TYPE DUT_HMI_06 :
STRUCT
	Manuals : DUT_HMI_06_MANUALS;
	ProductStatus 	: eProductStatus;
	State			: eStationState;
	EVDiagnostic 	: ARRAY[0..20] OF DUT_HMI_EV_Diagnostic;
	EVInfo			: ARRAY[0..CNC.NUM_MAX_MANUALS_06-1] OF DUT_HMI_EV_Info;
	Status			: USINT;
	CycleTime		: STRING;
	BroachTarget	: USINT;
END_STRUCT
END_TYPE

(* stored: Version 1.1.0.1, ProductVersion 3.1.4024.15
   DUT DUT_HMI_06: Id {afcf2016-aa5e-4288-b5d1-001be58b4a2d} *)
